TYPE T_NOTT_CRYO_STAT :
STRUCT
	//
	// Common attributes
	//
	bConfigured:	BOOL := FALSE;
	bSystemStarted:	BOOL := FALSE;	// Indicates if M_GetState has been called.

	bDone:			BOOL;			// Flag if controller is OK
	bBusy:			BOOL;			// Flag if controller is BUSY
	bError:			BOOL;			// Flag if controller is OK
	bActive:		BOOL;			// Flag if controller is ACTIVE
	
	nLastCommand:	E_NOTT_CRYO_CTRL_CMD 	:= E_NOTT_CRYO_CTRL_CMD.NONE;
	nState:			E_NOTT_CRYO_CTRL_STATE	:= E_NOTT_CRYO_CTRL_STATE.NONE;
	{attribute 'TcHmiSymbol.Show'}
	{attribute 'TcHmiSymbol.ReadOnly'}
	sState:			STRING(64);		// State as text


	//
	// PDS Cryo Controller specific attributes
	//
	
	// Simulation
	bSimulation:	BOOL := FALSE;	// If TRUE, System is simulated - Variant (V2_SIM)	
	bSim_RepressEnabled:	BOOL := FALSE;
	{attribute 'TcHmiSymbol.Show'}
	{attribute 'TcHmiSymbol.ReadOnly'}
	bVacuum:		BOOL := FALSE;
	{attribute 'TcHmiSymbol.Show'}
	{attribute 'TcHmiSymbol.ReadOnly'}		
	bVacuumOK:		BOOL := FALSE;		
	{attribute 'TcHmiSymbol.Show'}
	{attribute 'TcHmiSymbol.ReadOnly'}
	bPressureValid:	BOOL := FALSE;
	{attribute 'TcHmiSymbol.Show'}
	{attribute 'TcHmiSymbol.ReadOnly'}
	lrPressure_mbar:	LREAL;
	{attribute 'TcHmiSymbol.Show'}
	{attribute 'TcHmiSymbol.ReadOnly'}
	bCold:			BOOL := FALSE;	// Detector vote < cfg.lrTemp_Warm and cryostat is in vacuum
	{attribute 'TcHmiSymbol.Show'}
	{attribute 'TcHmiSymbol.ReadOnly'}
	bOP:			BOOL := FALSE;	// Detector/base-plate temperatures and VAGC pressure are operational

	bCoolantFlowOK:	BOOL := FALSE;		
	{attribute 'TcHmiSymbol.Show'}
	{attribute 'TcHmiSymbol.ReadOnly'}
	bHighestTempValid:	BOOL := FALSE;	// Highest temperature Valid flag
	{attribute 'TcHmiSymbol.Show'}
	{attribute 'TcHmiSymbol.ReadOnly'}
	bLowestTempValid:	BOOL := FALSE;	// Lowest temperature Valid flag
	{attribute 'TcHmiSymbol.Show'}
	{attribute 'TcHmiSymbol.ReadOnly'}
	lrHighestTempK:	LREAL;	// Highest temperature [K] in Cryostat
	{attribute 'TcHmiSymbol.Show'}
	{attribute 'TcHmiSymbol.ReadOnly'}
	lrLowestTempK:	LREAL;	// Lowest temperature [K] in Cryostat
	{attribute 'TcHmiSymbol.Show'}
	{attribute 'TcHmiSymbol.ReadOnly'}
	sLowestTempName:	STRING;
	{attribute 'TcHmiSymbol.Show'}
	{attribute 'TcHmiSymbol.ReadOnly'}
	sHighestTempName:	STRING;
	
	bIsPVPRunning:		BOOL := FALSE;
	bIsTMPRunning:		BOOL := FALSE;

END_STRUCT
END_TYPE

(* stored: Version 1.1.0.1, ProductVersion 3.1.4026.18
   DUT T_NOTT_CRYO_STAT: Id {e0babf34-620b-4f3b-9ccd-c42cad9ef3ae} *)
